INTERFACE I_Payload_A EXTENDS I_Payload

END_INTERFACE

(* stored: Version 1.1.0.1, ProductVersion 3.1.4024.2
   Itf I_Payload_A: Id {2c5c1cf3-5b02-47c9-adb4-4fba19f1e938} *)
